PROGRAM MAIN
VAR
END_VAR

END_PROGRAM

(* stored: Version 1.1.0.1
   POU MAIN: Id {0ca78153-12a1-425f-a0ef-fffe244bf1e5} *)
